// This function has been automatically generated from the project information.
{attribute 'signature_flag' := '1073741824'}
{attribute 'TcGenerated'}
{attribute 'no-analysis'}
FUNCTION F_GetTitle : WSTRING
VAR_INPUT
	
END_VAR

F_GetTitle := "Tc3_Base";

END_FUNCTION

(* stored: Version 1.1.0.1
   POU F_GetTitle: Id {a3a0a245-0bd9-4d13-a59c-8d9eadba71eb}, SpecialFunc None *)
